Staubli VAL3: CycleRefresh.pgx

program CycleRefresh()
  local num l_nEvent
  local num l_nSize[3]
  local num i
  local num l_nResult
  local bool l_bTrajRunning
begin
  // set the size
  call use:setSizeList(19,0,19,10)
  //
  // TRAJECTORY
  //
  if use:bUseRefresh
    // refresh the board
    call refreshStatic()
    //
    use:bUseRefresh=false
    //
    // rebuilt the Traj list
    //
    call refreshPoints(saveData:sTrajTypeUsing+" "+sTrajName)
    // look if the init has finished
    if cycleStatus:bSimulation
      nPoint=cycleStatus:nPoint
    endIf
    // REFRESH ACTUAL POINT
    use:nView=nPoint%use:nBottomY
    call use:listredraw(nPoint-use:nView)
  else
    // only update
    nPoint=cycleStatus:nPoint
    if use:nView>=nPoint%use:nBottomY
      // update the list
      use:nView=nPoint%use:nBottomY
      call use:listupdate(nPoint-use:nView)
    else
      //just the line
      call use:listcursor(use:nView,false)
      use:nView=nPoint%use:nBottomY
      call use:listcursor(use:nView,true)
    endIf
  endIf
end
